{attribute 'qualified_only'}
VAR_GLOBAL
	stAddCommand		: ST_AddCommand;
	stAddLongCommand	: ST_AddCommand;
	
	AddCommand1			: AddCommand 			:= (Val1 := 3, Val2 := 2);
	DelayedAddCommand1	: DelayedAddCommand 	:= (Val1 := 4, Val2 := 5);
END_VAR

(* stored: Version 1.1.0.1, ProductVersion 3.1.4022.10
   GVL Commands: Id {75e95b76-451e-476e-86cf-c478be106f96} *)
